# EPICS autosave request: iocBoot/ioc13idc/auto_positions.req
file "CARS_88_motor_positions.req", P=13IDC:
